												If there are more than 10 (DHP11B) or 64 (DHx41B) parameters to write, declare 
												NUMOF_INITIALPARAMETER in your program.
	
													VAR_GLOBAL CONSTANT
														NUMOF_INITIALPARAMETER : UDINT := 20;	
													END_VAR
	
												##################################################################*)
			-------------------------------------------------------------------------------------------------------------------------------------------------------------
		(* IDs of the PDO telegrams. The IDs are always calculated with the following IDs as a basis + the address of the bus coupler *)

		RxPDO 								ARRAY[1..32] OF MC_PDO_COSLAVE;			(* MOVI-PLC --> Slave *)
												(* := 16#200,16#300,16#400,16#500,16#780,16#240,16#340,16#440,16#540,16#7C0;	*)
		-------------------------------------------------------------------------------------------------------------------------------------------------------------
		TxPDO 								ARRAY[1..32] OF MC_PDO_COSLAVE; 			(* Slave --> MOVI-PLC *)
												(*:= 16#180,16#280,16#380,16#480,16#680,16#1C0,16#2C0,16#3C0,16#4C0,16#6C0;*)
	*)
END_VAR
IF Enable AND NOT Done THEN

	(*########################################################

		Configuration of CANopenSlave (SEW OCC11B)
		
	#########################################################

		TransmissionType for TxPDOs and RxPDOs:

			0:										Event controlled and sychron (with SYNC-Object)
			1-240:									Cyclic and synchron (with SYNC-Object)
			254:									Producer specified
			255:									Acyclic and eventcontrolled 
			255 and EventTime = InhibitTime:	Cyclic

	#########################################################	*)


	(*************************************************** TxPDOs of CANOpenSlave ( MOVI-PLC ReceiveObjects) ***********************************************************)

	ExtConfig.NumberOfTxPDO				:= 4;		(*  TxPDO ---> CANopenSlave Transmit *)

	ExtConfig.TxPDO[1].EventTime			:= 200;		(* Slave: Index 0x18xx SubIndex 5: CycleTime in ms for CANopenSlave TXPDO *)
	ExtConfig.TxPDO[1].InhibitTime			:= 5;		(* Slave: Index 0x18xx SubIndex 3: InhibitTime in ms for CANopenSlave TxPDO *)
	ExtConfig.TxPDO[1].TransmissionType	:= 255;		(* Slave: Index 0x18xx SubIndex 2: TransmissionType for this TxPDO *)

	ExtConfig.TxPDO[2].EventTime			:= 100;		(* Slave: Index 0x18xx SubIndex 5: CycleTime in ms for CANopenSlave TXPDO *)
	ExtConfig.TxPDO[2].InhibitTime			:= 100;		(* Slave: Index 0x18xx SubIndex 3: InhibitTime in ms for CANopenSlave TxPDO *)
	ExtConfig.TxPDO[2].TransmissionType	:= 255;		(* Slave: Index 0x18xx SubIndex 2: TransmissionType for this TxPDO *)

	ExtConfig.TxPDO[3].EventTime			:= 100;		(* Slave: Index 0x18xx SubIndex 5: CycleTime in ms for CANopenSlave TXPDO *)
	ExtConfig.TxPDO[3].InhibitTime			:= 100;		(* Slave: Index 0x18xx SubIndex 3: InhibitTime in ms for CANopenSlave TxPDO *)
	ExtConfig.TxPDO[3].TransmissionType	:= 255;		(* Slave: Index 0x18xx SubIndex 2: TransmissionType for this TxPDO *)

	ExtConfig.TxPDO[4].EventTime			:= 100;		(* Slave: Index 0x18xx SubIndex 5: CycleTime in ms for CANopenSlave TXPDO *)
	ExtConfig.TxPDO[4].InhibitTime			:= 100;		(* Slave: Index 0x18xx SubIndex 3: InhibitTime in ms for CANopenSlave TxPDO *)
	ExtConfig.TxPDO[4].TransmissionType	:= 255;		(* Slave: Index 0x18xx SubIndex 2: TransmissionType for this TxPDO *)


	(*************************************************** RxPDOs of CANOpenSlave ( MOVI-PLC TransmitObjects) **********************************************************)

	ExtConfig.NumberOfRxPDO				:= 4;		(*  RxPDO ---> CANopenSlave Receive *)

	ExtConfig.RxPDO[1].EventTime			:= 200;		(* Master: CycleTime in ms for TransmitObjects (MOVI-PLC) *)
	ExtConfig.RxPDO[1].InhibitTime			:= 5;		(* Master: InhibitTime in ms for TransmitObjects (MOVI-PLC) *)
	ExtConfig.RxPDO[1].Length				:= 1;		(* Master: Length of this TransmitObject in bytes *)
	ExtConfig.RxPDO[1].TransmissionType	:= 255;		(* Slave: Index 0x14xx SubIndex 2: TransmissionType for this RxPDO *)

	ExtConfig.RxPDO[2].EventTime			:= 100;		(* Master: CycleTime in ms for TransmitObjects (MOVI-PLC) *)
	ExtConfig.RxPDO[2].InhibitTime			:= 100;		(* Master: InhibitTime in ms for TransmitObjects (MOVI-PLC) *)
	ExtConfig.RxPDO[2].Length				:= 8;		(* Master: Length of this TransmitObject in bytes *)
	ExtConfig.RxPDO[2].TransmissionType	:= 255;		(* Slave: Index 0x14xx SubIndex 2: TransmissionType for this RxPDO *)

	ExtConfig.RxPDO[3].EventTime			:= 100;		(* Master: CycleTime in ms for TransmitObjects (MOVI-PLC) *)
	ExtConfig.RxPDO[3].InhibitTime			:= 100;		(* Master: InhibitTime in ms for TransmitObjects (MOVI-PLC) *)
	ExtConfig.RxPDO[3].Length				:= 8;		(* Master: Length of this TransmitObject in bytes *)
	ExtConfig.RxPDO[3].TransmissionType	:= 255;		(* Slave: Index 0x14xx SubIndex 2: TransmissionType for this RxPDO *)

	ExtConfig.RxPDO[4].EventTime			:= 100;		(* Master: CycleTime in ms for TransmitObjects (MOVI-PLC) *)
	ExtConfig.RxPDO[4].InhibitTime			:= 100;		(* Master: InhibitTime in ms for TransmitObjects (MOVI-PLC) *)
	ExtConfig.RxPDO[4].Length				:= 8;		(* Master: Length of this TransmitObject in bytes *)
	ExtConfig.RxPDO[4].TransmissionType	:= 255;		(* Slave: Index 0x14xx SubIndex 2: TransmissionType for this RxPDO *)


	(***************************************************** Additional parameters to set in the CANOpenSlave  ***************************************************************)

	(* Enable transmission of analog inputs *)
	ExtConfig.stInitialParameter_COSlave.aIndex[1]			:= 16#6423;
	ExtConfig.stInitialParameter_COSlave.aSubIndex[1]	:= 0;
	ExtConfig.stInitialParameter_COSlave.aBytes[1]		:= 1;
	ExtConfig.stInitialParameter_COSlave.aData[1]			:= 1;


	(********************************************** Additional configuration. Default values are in most cases sufficient *****************************************************)

	ExtConfig.bIOHold						:= FALSE;
	ExtConfig.bNoSettingsDownload			:= FALSE;
	ExtConfig.bWaitBeforeOperational		:= FALSE;
	ExtConfig.bResetUnconditional			:= FALSE;

	ExtConfig.TimeOutHeartBeat				:= 400;				(* [ms] *)
	ExtConfig.TimeOutNodeGuarding		:= 0;				(* [ms]. CAUTION ! DHP11B (MOVI-PLC basic) does NOT support NodeGuarding *)
	ExtConfig.TimeOutInitSequence			:= 10;				(* [seconds]. If the Init-Sequence takes longer than this TimeOut time --> Error *)
	ExtConfig.SyncCOBID						:= 0;				(* SyncObject ID for TransmissionType 0-240 (RxPDO). Usually 16#8000_0080. If 0, the ID will not be written *)
	ExtConfig.SyncTime						:= 0;				(* CycleTime for the SYNC-Object *)

	ExtConfig.SBUSGateway_Address			:= 0(*1001*);			(* OSC71B Address,when used *)

	ExtConfig.TxPDO[1].COBID				:= 16#180;			(* In order to disable the use of RTR frames for the PDOs, set bit 30 = "RTR not allowed" *)
	ExtConfig.TxPDO[2].COBID				:= 16#280;			(* Ex. 16#4000_0280 *)
	ExtConfig.TxPDO[3].COBID				:= 16#380;
	ExtConfig.TxPDO[4].COBID				:= 16#480;			(* NOTE! These values are base values. The input "Address" will automatically be added *)
	ExtConfig.TxPDO[5].COBID				:= 16#680;
	ExtConfig.TxPDO[6].COBID				:= 16#1C0;
	ExtConfig.TxPDO[7].COBID				:= 16#2C0;
	ExtConfig.TxPDO[8].COBID				:= 16#3C0;
	ExtConfig.TxPDO[9].COBID				:= 16#4C0;
	ExtConfig.TxPDO[10].COBID				:= 16#6C0;

	ExtConfig.RxPDO[1].COBID				:= 16#200;
	ExtConfig.RxPDO[2].COBID				:= 16#300;
	ExtConfig.RxPDO[3].COBID				:= 16#400;
	ExtConfig.RxPDO[4].COBID				:= 16#500;
	ExtConfig.RxPDO[5].COBID				:= 16#780;
	ExtConfig.RxPDO[6].COBID				:= 16#240;
	ExtConfig.RxPDO[7].COBID				:= 16#340;
	ExtConfig.RxPDO[8].COBID				:= 16#440;
	ExtConfig.RxPDO[9].COBID				:= 16#540;
	ExtConfig.RxPDO[10].COBID				:= 16#7C0;

	Done := TRUE;

END_IF
END_FUNCTION_BLOCK

(* POU CodeSamples/CANopen/UniversalMaster/FB_Configuration_CANopenSlave_TR_AbsEncoder, ST *)
FUNCTION_BLOCK FB_Configuration_CANopenSlave_TR_AbsEncoder
VAR_INPUT
	Enable: BOOL; 			(* Activate config *)
END_VAR
VAR_OUTPUT
	Done: BOOL;				(* Config done *)
END_VAR
VAR_IN_OUT
	ExtConfig : MC_EXTENDEDCONFIG_COSLAVE	;
	(*
		########################################################################################################
			MC_EXTENDEDCONFIG_COSLAVE
		#########################################################################################################

						
		Variable								Value			Description
		-------------------------------------------------------------------------------------------------------------------------------------------------------------
		bWaitBeforeOperational 				BOOL;			When TRUE, after the coupler has been parameterized, it won't be switched in operational
																before this variable is FALSE. This can be used for example, to store the configuration with the FB
																MPLC_Universal_CANopen, with Service "SEWIOS_STORE", after a reset of the coppler 
		-------------------------------------------------------------------------------------------------------------------------------------------------------------
		bNoSettingsDownload 				BOOL;			TRUE : No configuration of the module. The configuration has to be done manually.
		-------------------------------------------------------------------------------------------------------------------------------------------------------------
		bResetUnconditional 					BOOL;			Even if the Connect FB isn't in fault it is possible to reset the bus coppler
		-------------------------------------------------------------------------------------------------------------------------------------------------------------
		bIOHold 								BOOL;			TRUE : Input data remain unchanged and the output data are not resetet also if the FB is in fault 
		-------------------------------------------------------------------------------------------------------------------------------------------------------------
		TimeOutHeartBeat					UINT;			If this value (ms) is different to zero, HeartbeatMode will be activated
		-------------------------------------------------------------------------------------------------------------------------------------------------------------
		TimeOutNodeGuarding 				UINT;			If this value (ms) is different to zero, NodeGuarding will be activated. 
																Caution ! The MOVI-PLC basic doesn´t support NodeGuarding 
		-------------------------------------------------------------------------------------------------------------------------------------------------------------
		TimeOutInitSequence					UINT;			Timeout for initialisation sequence (seconds) 
		-------------------------------------------------------------------------------------------------------------------------------------------------------------
		NumberOfRxPDO 					UINT;			Receive PDO : MOVI-PLC --> Slave  max. 32 
		-------------------------------------------------------------------------------------------------------------------------------------------------------------
		NumberOfTxPDO 						UINT;			Send PDO :      Slave --> MOVI-PLC  max 32 
		-------------------------------------------------------------------------------------------------------------------------------------------------------------	
		SyncTime 								USINT;			Cycle time of the sync telegram in ms. 
																Default = 0 : no sync will be started.
																If  SyncTime > 0, this FB initializes a sync telegram with the ID set at SyncCOBID. 
																The slave has to support synchronous communication 
		-------------------------------------------------------------------------------------------------------------------------------------------------------------
		SyncCOBID							UINT;			Index 1005h. ID of the sync telegram. Usually 16#80. IF 0, the ID won't be written.
		-------------------------------------------------------------------------------------------------------------------------------------------------------------
		SyncTimeOut 							INT := -1;		Index 1006h. Normally equal to SyncTime. 
																The slave usually set SyncTimeOut equal to SyncTime * 1.5. 
																If < 0, the index won't be written. 0 means no control over the sync interval 
		-------------------------------------------------------------------------------------------------------------------------------------------------------------
		stInitialParameter_COSlave 			MC_INITIALPARAMETER_COSLAVE;
												(*#################################################################
												With this struct, user defined parameters will be written to the BusCoupler after the
												initialization of the MPLC_ConnectUniversalSlave_CANopen. 
												Add the following code to your program to initialise the struct : 
												Example:
												Index 16#6423:	Activates the event-driven transmission of PDOs with analog inputs
												Index 16#3500:	Index from the manufacturer specific profile area
	
													stInitialParameter_COSlave.aIndex[1] := 16#6423;  	(* Index to write to *)
													stInitialParameter_COSlave.aSubIndex[1] := 0;   	(* SubIndex to write to *)
													stInitialParameter_COSlave.aBytes[1] := 1;   		(* Number of bytes to write  *)
													stInitialParameter_COSlave.aData[1] := 1;   			(* Data *)
	
													stInitialParameter_COSlave.aIndex[2] := 16#3500;  	(* Index to write to *)
													stInitialParameter_COSlave.aSubIndex[2] := 0;   	(* SubIndex to write to *)
													stInitialParameter_COSlave.aBytes[2] := 2;   		(* Number of bytes to write *)
													stInitialParameter_COSlave.aData[2] := 5;   			(* Data *)
	
												If there are more than 10 (DHP11B) or 64 (DHx41B) parameters to write, declare 
												NUMOF_INITIALPARAMETER in your program.
	
													VAR_GLOBAL CONSTANT
														NUMOF_INITIALPARAMETER : UDINT := 20;	
													END_VAR
	
												##################################################################*)
			-------------------------------------------------------------------------------------------------------------------------------------------------------------
		(* IDs of the PDO telegrams. The IDs are always calculated with the following IDs as a basis + the address of the bus coupler *)

		RxPDO 								ARRAY[1..32] OF MC_PDO_COSLAVE;			(* MOVI-PLC --> Slave *)
												(* := 16#200,16#300,16#400,16#500,16#780,16#240,16#340,16#440,16#540,16#7C0;	*)
		-------------------------------------------------------------------------------------------------------------------------------------------------------------
		TxPDO 								ARRAY[1..32] OF MC_PDO_COSLAVE; 			(* Slave --> MOVI-PLC *)
												(*:= 16#180,16#280,16#380,16#480,16#680,16#1C0,16#2C0,16#3C0,16#4C0,16#6C0;*)
	*)
END_VAR
IF Enable AND NOT Done THEN

	(*########################################################

		Configuration of CANopenSlave (T+R AbsEncoder)
		
	#########################################################

		TransmissionType for TxPDOs and RxPDOs:

			0:										Event controlled and sychron (with SYNC-Object)
			1-240:									Cyclic and synchron (with SYNC-Object)
			254:									Producer specified
			255:									Acyclic and eventcontrolled 
			255 and EventTime = InhibitTime:	Cyclic

	#########################################################	*)


	(*************************************************** TxPDOs of CANOpenSlave ( MOVI-PLC ReceiveObjects) ***********************************************************)

	ExtConfig.NumberOfTxPDO				:= 1;		(*  TxPDO ---> CANopenSlave Transmit *)

	ExtConfig.TxPDO[1].EventTime			:= 20;		(* Slave: Index 0x18xx SubIndex 5: CycleTime in ms for CANopenSlave TXPDO *)
	ExtConfig.TxPDO[1].InhibitTime			:= 20;		(* Slave: Index 0x18xx SubIndex 3: InhibitTime in ms for CANopenSlave TxPDO *)
	ExtConfig.TxPDO[1].TransmissionType	:= 254;		(* Slave: Index 0x18xx SubIndex 2: TransmissionType for this TxPDO *)


	(*************************************************** RxPDOs of CANOpenSlave ( MOVI-PLC TransmitObjects) **********************************************************)

	ExtConfig.NumberOfRxPDO				:= 0;		(*  RxPDO ---> CANopenSlave Receive *)

	(* ExtConfig.RxPDO[1].EventTime		:= 0;		(* Master: CycleTime in ms for TransmitObjects (MOVI-PLC) *)
	ExtConfig.RxPDO[1].InhibitTime			:= 0;		(* Master: InhibitTime in ms for TransmitObjects (MOVI-PLC) *)
	ExtConfig.RxPDO[1].Length				:= 2;		(* Master: Length of this TransmitObject in bytes *)
	ExtConfig.RxPDO[1].TransmissionType	:= 255;		(* Slave: Index 0x14xx SubIndex 2: TransmissionType for this RxPDO *)*)


	(***************************************************** Additional parameters to set in the CANOpenSlave  ***************************************************************)

	(* Set rotation direction *)
	ExtConfig.stInitialParameter_COSlave.aIndex[1]			:= 16#6000;
	ExtConfig.stInitialParameter_COSlave.aSubIndex[1]	:= 0;
	ExtConfig.stInitialParameter_COSlave.aBytes[1]		:= 2;
	ExtConfig.stInitialParameter_COSlave.aData[1]			:= 0;		(* 0 = CV, 1 = CCV *)

	(* Set cyclic timer for Tx PDO1 *)
	ExtConfig.stInitialParameter_COSlave.aIndex[2]			:= 16#6200;
	ExtConfig.stInitialParameter_COSlave.aSubIndex[2]	:= 0;
	ExtConfig.stInitialParameter_COSlave.aBytes[2]		:= 2;
	ExtConfig.stInitialParameter_COSlave.aData[2]			:= 20;		(* [ms] *)

	(* Write reference offset to AbsEncoder, Index 6003.0, data = new position *)
	(* Write Delivery state to AbsEncoder, Index 1011.1, data = 16#6C_6F_61_64 (load) *)
	(* Save values in Flash memory in the AbsEncoder, Index 1010.1, data = 16#73_61_76_65 (save) *)


	(********************************************** Additional configuration. Default values are in most cases sufficient *****************************************************)

	ExtConfig.bIOHold						:= FALSE;
	ExtConfig.bNoSettingsDownload			:= FALSE;
	ExtConfig.bWaitBeforeOperational		:= FALSE;
	ExtConfig.bResetUnconditional			:= FALSE;

	ExtConfig.TimeOutHeartBeat				:= 0;				(* [ms] *)
	ExtConfig.TimeOutNodeGuarding		:= 400;				(* [ms]. CAUTION ! DHP11B (MOVI-PLC basic) does NOT support NodeGuarding *)
	ExtConfig.TimeOutInitSequence			:= 5;				(* [seconds]. If the Init-Sequence takes longer than this TimeOut time --> Error *)
	ExtConfig.SyncCOBID						:= 0;				(* SyncObject ID for TransmissionType 0-240 (RxPDO). Usually 128. If 0, the ID will not be written *)
	ExtConfig.SyncTime						:= 0;				(* CycleTime for the SYNC-Object *)

	ExtConfig.TxPDO[1].COBID				:= 16#180;			(* In order to disable the use of RTR frames for the PDOs, set bit 30 = "RTR not allowed" *)
	ExtConfig.TxPDO[2].COBID				:= 16#280;			(* Ex. 16#4000_0280 *)
	ExtConfig.TxPDO[3].COBID				:= 16#380;
	ExtConfig.TxPDO[4].COBID				:= 16#480;			(* NOTE! These values are base values. The input "Address" will automatically be added *)
	ExtConfig.TxPDO[5].COBID				:= 16#680;
	ExtConfig.TxPDO[6].COBID				:= 16#1C0;
	ExtConfig.TxPDO[7].COBID				:= 16#2C0;
	ExtConfig.TxPDO[8].COBID				:= 16#3C0;
	ExtConfig.TxPDO[9].COBID				:= 16#4C0;
	ExtConfig.TxPDO[10].COBID				:= 16#6C0;

	ExtConfig.RxPDO[1].COBID				:= 16#200;
	ExtConfig.RxPDO[2].COBID				:= 16#300;
	ExtConfig.RxPDO[3].COBID				:= 16#400;
	ExtConfig.RxPDO[4].COBID				:= 16#500;
	ExtConfig.RxPDO[5].COBID				:= 16#780;
	ExtConfig.RxPDO[6].COBID				:= 16#240;
	ExtConfig.RxPDO[7].COBID				:= 16#340;
	ExtConfig.RxPDO[8].COBID				:= 16#440;
	ExtConfig.RxPDO[9].COBID				:= 16#540;
	ExtConfig.RxPDO[10].COBID				:= 16#7C0;

	Done := TRUE;

END_IF
END_FUNCTION_BLOCK

(* POU CodeSamples/CANopen/UniversalMaster/FB_Configuration_CANopenSlave_Wachendorff, ST *)
FUNCTION_BLOCK FB_Configuration_CANopenSlave_Wachendorff
VAR_INPUT
	Enable: BOOL; 			(* Activate config *)
END_VAR
VAR_OUTPUT
	Done: BOOL;				(* Config done *)
END_VAR
VAR_IN_OUT
	ExtConfig : MC_EXTENDEDCONFIG_COSLAVE	;
	(*
		########################################################################################################
			MC_EXTENDEDCONFIG_COSLAVE
		#########################################################################################################

						
		Variable								Value			Description
		-------------------------------------------------------------------------------------------------------------------------------------------------------------
		bWaitBeforeOperational 				BOOL;			When TRUE, after the coupler has been parameterized, it won't be switched in operational
																before this variable is FALSE. This can be used for example, to store the configuration with the FB
																MPLC_Universal_CANopen, with Service "SEWIOS_STORE", after a reset of the coppler 
		-------------------------------------------------------------------------------------------------------------------------------------------------------------
		bNoSettingsDownload 				BOOL;			TRUE : No configuration of the module. The configuration has to be done manually.
		-------------------------------------------------------------------------------------------------------------------------------------------------------------
		bResetUnconditional 					BOOL;			Even if the Connect FB isn't in fault it is possible to reset the bus coppler
		-------------------------------------------------------------------------------------------------------------------------------------------------------------
		bIOHold 								BOOL;			TRUE : Input data remain unchanged and the output data are not resetet also if the FB is in fault 
		-------------------------------------------------------------------------------------------------------------------------------------------------------------
		TimeOutHeartBeat					UINT;			If this value (ms) is different to zero, HeartbeatMode will be activated

		bNoHeartBeat_Producer:				BOOL := FALSE; (*Index 1017 SubIndex 0 not available *)
		-------------------------------------------------------------------------------------------------------------------------------------------------------------
		TimeOutNodeGuarding 				UINT;			If this value (ms) is different to zero, NodeGuarding will be activated. 
																Caution ! The MOVI-PLC basic doesn´t support NodeGuarding 
	
		bNoNodeGuarding:					BOOL:=FALSE; (* the Index of NodeGuarding isn`t available *)
		-------------------------------------------------------------------------------------------------------------------------------------------------------------
		TimeOutInitSequence					UINT;			Timeout for initialisation sequence (seconds) 
		-------------------------------------------------------------------------------------------------------------------------------------------------------------
		NumberOfRxPDO 					UINT;			Receive PDO : MOVI-PLC --> Slave  max. 32 
		-------------------------------------------------------------------------------------------------------------------------------------------------------------
		NumberOfTxPDO 						UINT;			Send PDO :      Slave --> MOVI-PLC  max 32 
		-------------------------------------------------------------------------------------------------------------------------------------------------------------	
		OffsetOfRxPDO:						UINT;			Offset for the 1. RxPDO
		-------------------------------------------------------------------------------------------------------------------------------------------------------------		
		OffsetOfTxPDO:						UINT;			Offset for the 1. TxPDO
		-------------------------------------------------------------------------------------------------------------------------------------------------------------	
		SyncTime 								USINT;			Cycle time of the sync telegram in ms. 
																Default = 0 : no sync will be started.
																If  SyncTime > 0, this FB initializes a sync telegram with the ID set at SyncCOBID. 
																The slave has to support synchronous communication 
		-------------------------------------------------------------------------------------------------------------------------------------------------------------
		SyncCOBID							UINT;			Index 1005h. ID of the sync telegram. Usually 16#80. IF 0, the ID won't be written.
		-------------------------------------------------------------------------------------------------------------------------------------------------------------
		SyncTimeOut 							INT := -1;		Index 1006h. Normally equal to SyncTime. 
																The slave usually set SyncTimeOut equal to SyncTime * 1.5. 
																If < 0, the index won't be written. 0 means no control over the sync interval 
		-------------------------------------------------------------------------------------------------------------------------------------------------------------
		stInitialParameter_COSlave 			MC_INITIALPARAMETER_COSLAVE;
												(*#################################################################
												With this struct, user defined parameters will be written to the BusCoupler after the
												initialization of the MPLC_ConnectUniversalSlave_CANopen. 
												Add the following code to your program to initialise the struct : 
												Example:
												Index 16#6423:	Activates the event-driven transmission of PDOs with analog inputs
												Index 16#3500:	Index from the manufacturer specific profile area
	
													stInitialParameter_COSlave.aIndex[1] := 16#6423;  	(* Index to write to *)
													stInitialParameter_COSlave.aSubIndex[1] := 0;   	(* SubIndex to write to *)
													stInitialParameter_COSlave.aBytes[1] := 1;   		(* Number of bytes to write  *)
													stInitialParameter_COSlave.aData[1] := 1;   			(* Data *)
	
													stInitialParameter_COSlave.aIndex[2] := 16#3500;  	(* Index to write to *)
													stInitialParameter_COSlave.aSubIndex[2] := 0;   	(* SubIndex to write to *)
													stInitialParameter_COSlave.aBytes[2] := 2;   		(* Number of bytes to write *)
													stInitialParameter_COSlave.aData[2] := 5;   			(* Data *)
	
												If there are more than 10 (DHP11B) or 64 (DHx41B) parameters to write, declare 
												NUMOF_INITIALPARAMETER in your program.
	
													VAR_GLOBAL CONSTANT
														NUMOF_INITIALPARAMETER : UDINT := 20;	
													END_VAR
	
												##################################################################*)

		bNoDeactivatePDO:			BOOL := FALSE; (* Change of Transmission Type, Inhibit- and Event- Time without deactivate RxPDO and TxPDO*)

			-------------------------------------------------------------------------------------------------------------------------------------------------------------
		(* IDs of the PDO telegrams. The IDs are always calculated with the following IDs as a basis + the address of the bus coupler *)

		RxPDO 								ARRAY[1..32] OF MC_PDO_COSLAVE;			(* MOVI-PLC --> Slave *)
												(* := 16#200,16#300,16#400,16#500,16#780,16#240,16#340,16#440,16#540,16#7C0;	*)
		-------------------------------------------------------------------------------------------------------------------------------------------------------------
		TxPDO 								ARRAY[1..32] OF MC_PDO_COSLAVE; 			(* Slave --> MOVI-PLC *)
												(*:= 16#180,16#280,16#380,16#480,16#680,16#1C0,16#2C0,16#3C0,16#4C0,16#6C0;*)
	*)
END_VAR
{library private}
VAR
	fbCANopen_aktiv: CANopen_activ;
	Error: BOOL;
	Error_ID: DINT;
END_VAR
IF Enable AND NOT Done THEN

(*  !!!!!!!  only once TO activate !!!!!!*)
(*
	(*######################################################*)
		(* set Baudrate and CAN-ID *)
	fbCANopen_aktiv(Node:= SBUS_Node_2,
					Address_Default := 60,(* Default Address or old Address 0...127*)
					Address:= 60,(* new Address 1...63*)
					Baudrate:=2, (* 0 = 1 M , 2 = 500 k , 3 = 250 k baud*)
					Error => Error,
					ErrorID=> Error_ID);


		RETURN;
	(*######################################################*)
*)


	(*########################################################

		Configuration of CANopenSlave (Wachendorff AbsEncoder)
		
	#########################################################

		TransmissionType for TxPDOs and RxPDOs:

			0:										Event controlled and sychron (with SYNC-Object)
			1-240:									Cyclic and synchron (with SYNC-Object)
			254:									Producer specified
			255:									Acyclic and eventcontrolled 
			255 and EventTime = InhibitTime:	Cyclic

	#########################################################	*)

(*	ExtConfig.OffsetOfTxPDO := 2;*)
	(*************************************************** TxPDOs of CANOpenSlave ( MOVI-PLC ReceiveObjects) ***********************************************************)

	ExtConfig.NumberOfTxPDO				:= 3;		(*  TxPDO ---> CANopenSlave Transmit *)

	ExtConfig.TxPDO[1].EventTime			:= 20;		(* Slave: Index 0x18xx SubIndex 5: CycleTime in ms for CANopenSlave TXPDO *)
	ExtConfig.TxPDO[1].InhibitTime			:= 10;		(* Slave: Index 0x18xx SubIndex 3: InhibitTime in ms for CANopenSlave TxPDO *)
	ExtConfig.TxPDO[1].TransmissionType	:= 254;		(* Slave: Index 0x18xx SubIndex 2: TransmissionType for this TxPDO *)

	ExtConfig.TxPDO[2].EventTime			:= 0;		(* Slave: Index 0x18xx SubIndex 5: CycleTime in ms for CANopenSlave TXPDO *)
	ExtConfig.TxPDO[2].InhibitTime			:= 0;		(* Slave: Index 0x18xx SubIndex 3: InhibitTime in ms for CANopenSlave TxPDO *)
	ExtConfig.TxPDO[2].TransmissionType	:= 1;		(* Slave: Index 0x18xx SubIndex 2: TransmissionType for this TxPDO *)

	ExtConfig.TxPDO[3].EventTime			:= 0;		(* Slave: Index 0x18xx SubIndex 5: CycleTime in ms for CANopenSlave TXPDO *)
	ExtConfig.TxPDO[3].InhibitTime			:= 0;		(* Slave: Index 0x18xx SubIndex 3: InhibitTime in ms for CANopenSlave TxPDO *)
	ExtConfig.TxPDO[3].TransmissionType	:= 1;		(* Slave: Index 0x18xx SubIndex 2: TransmissionType for this TxPDO *)

	(*************************************************** RxPDOs of CANOpenSlave ( MOVI-PLC TransmitObjects) **********************************************************)

	ExtConfig.NumberOfRxPDO				:= 0;		(*  RxPDO ---> CANopenSlave Receive *)

	(* ExtConfig.RxPDO[1].EventTime		:= 0;		(* Master: CycleTime in ms for TransmitObjects (MOVI-PLC) *)
	ExtConfig.RxPDO[1].InhibitTime			:= 0;		(* Master: InhibitTime in ms for TransmitObjects (MOVI-PLC) *)
	ExtConfig.RxPDO[1].Length				:= 2;		(* Master: Length of this TransmitObject in bytes *)
	ExtConfig.RxPDO[1].TransmissionType	:= 255;		(* Slave: Index 0x14xx SubIndex 2: TransmissionType for this RxPDO *)*)


	(***************************************************** Additional parameters to set in the CANOpenSlave  ***************************************************************)

	(* Set rotation direction *)
	ExtConfig.stInitialParameter_COSlave.aIndex[1]			:= 16#6000;
	ExtConfig.stInitialParameter_COSlave.aSubIndex[1]	:= 0;
	ExtConfig.stInitialParameter_COSlave.aBytes[1]		:= 2;
	ExtConfig.stInitialParameter_COSlave.aData[1]			:= 0;		(* 0 = CV, 1 = CCV *)

(*	(* Set cyclic timer for Tx PDO1 *)
	ExtConfig.stInitialParameter_COSlave.aIndex[2]			:= 16#6200;
	ExtConfig.stInitialParameter_COSlave.aSubIndex[2]	:= 0;
	ExtConfig.stInitialParameter_COSlave.aBytes[2]		:= 2;
	ExtConfig.stInitialParameter_COSlave.aData[2]			:= 20;		(* [ms] *)*)

(* deactivate Tx PDO1 *)
	ExtConfig.stInitialParameter_COSlave.aIndex[2]			:= 16#1800;
	ExtConfig.stInitialParameter_COSlave.aSubIndex[2]	:= 2;
	ExtConfig.stInitialParameter_COSlave.aBytes[2]		:= 1;
	ExtConfig.stInitialParameter_COSlave.aData[2]			:= 16#FF;

	ExtConfig.stInitialParameter_COSlave.aIndex[3]			:= 16#1800;
	ExtConfig.stInitialParameter_COSlave.aSubIndex[3]	:= 5;
	ExtConfig.stInitialParameter_COSlave.aBytes[3]		:= 2;
	ExtConfig.stInitialParameter_COSlave.aData[3]			:= 16#0000;

(* deactivate Tx PDO2 *)
	ExtConfig.stInitialParameter_COSlave.aIndex[4]			:= 16#1801;
	ExtConfig.stInitialParameter_COSlave.aSubIndex[4]	:= 2;
	ExtConfig.stInitialParameter_COSlave.aBytes[4]		:= 1;
	ExtConfig.stInitialParameter_COSlave.aData[4]			:= 16#FF;

	ExtConfig.stInitialParameter_COSlave.aIndex[5]			:= 16#1801;
	ExtConfig.stInitialParameter_COSlave.aSubIndex[5]	:= 5;
	ExtConfig.stInitialParameter_COSlave.aBytes[5]		:= 2;
	ExtConfig.stInitialParameter_COSlave.aData[5]			:= 16#0000;

	(* Write reference offset to AbsEncoder, Index 6003.0, data = new position *)
	(* Write Delivery state to AbsEncoder, Index 1011.1, data = 16#6C_6F_61_64 (load) *)
	(* Save values in Flash memory in the AbsEncoder, Index 1010.1, data = 16#73_61_76_65 (save) *)


	(********************************************** Additional configuration. Default values are in most cases sufficient *****************************************************)

	ExtConfig.bIOHold						:= FALSE;
	ExtConfig.bNoSettingsDownload			:= FALSE;
	ExtConfig.bWaitBeforeOperational		:= FALSE;
	ExtConfig.bResetUnconditional			:= FALSE;

	ExtConfig.TimeOutHeartBeat				:= 400;				(* [ms] *)
	ExtConfig.TimeOutNodeGuarding		:= 0;				(* [ms]. CAUTION ! DHP11B (MOVI-PLC basic) does NOT support NodeGuarding *)
	ExtConfig.TimeOutInitSequence			:= 15;				(* [seconds]. If the Init-Sequence takes longer than this TimeOut time --> Error *)
	ExtConfig.SyncCOBID						:= 128;				(* SyncObject ID for TransmissionType 0-240 (RxPDO). Usually 128. If 0, the ID will not be written *)
	ExtConfig.SyncTime						:= 5;				(* CycleTime for the SYNC-Object *)

	ExtConfig.TxPDO[1].COBID				:= 16#180;			(* In order to disable the use of RTR frames for the PDOs, set bit 30 = "RTR not allowed" *)
	ExtConfig.TxPDO[2].COBID				:= 16#280;			(* Ex. 16#4000_0280 *)
	ExtConfig.TxPDO[3].COBID				:= 16#380;
	ExtConfig.TxPDO[4].COBID				:= 16#480;			(* NOTE! These values are base values. The input "Address" will automatically be added *)
	ExtConfig.TxPDO[5].COBID				:= 16#680;
	ExtConfig.TxPDO[6].COBID				:= 16#1C0;
	ExtConfig.TxPDO[7].COBID				:= 16#2C0;
	ExtConfig.TxPDO[8].COBID				:= 16#3C0;
	ExtConfig.TxPDO[9].COBID				:= 16#4C0;
	ExtConfig.TxPDO[10].COBID				:= 16#6C0;

	ExtConfig.RxPDO[1].COBID				:= 16#200;
	ExtConfig.RxPDO[2].COBID				:= 16#300;
	ExtConfig.RxPDO[3].COBID				:= 16#400;
	ExtConfig.RxPDO[4].COBID				:= 16#500;
	ExtConfig.RxPDO[5].COBID				:= 16#780;
	ExtConfig.RxPDO[6].COBID				:= 16#240;
	ExtConfig.RxPDO[7].COBID				:= 16#340;
	ExtConfig.RxPDO[8].COBID				:= 16#440;
	ExtConfig.RxPDO[9].COBID				:= 16#540;
	ExtConfig.RxPDO[10].COBID				:= 16#7C0;

	Done := TRUE;
END_IF
END_FUNCTION_BLOCK

(* POU CodeSamples/CANopen/UniversalMaster/FB_Configuration_CANopenSlave_WAGO_750_337, ST *)
FUNCTION_BLOCK FB_Configuration_CANopenSlave_WAGO_750_337
VAR_INPUT
	Enable: BOOL; 			(* Activate config *)
END_VAR
VAR_OUTPUT
	Done: BOOL;				(* Config done *)
END_VAR
VAR_IN_OUT
	ExtConfig : MC_EXTENDEDCONFIG_COSLAVE	;
	(*
		########################################################################################################
			MC_EXTENDEDCONFIG_COSLAVE
		#########################################################################################################

						
		Variable								Value			Description
		-------------------------------------------------------------------------------------------------------------------------------------------------------------
		bWaitBeforeOperational 				BOOL;			When TRUE, after the coupler has been parameterized, it won't be switched in operational
																before this variable is FALSE. This can be used for example, to store the configuration with the FB
																MPLC_Universal_CANopen, with Service "SEWIOS_STORE", after a reset of the coppler 
		-------------------------------------------------------------------------------------------------------------------------------------------------------------
		bNoSettingsDownload 				BOOL;			TRUE : No configuration of the module. The configuration has to be done manually.
		-------------------------------------------------------------------------------------------------------------------------------------------------------------
		bResetUnconditional 					BOOL;			Even if the Connect FB isn't in fault it is possible to reset the bus coppler
		-------------------------------------------------------------------------------------------------------------------------------------------------------------
		bIOHold 								BOOL;			TRUE : Input data remain unchanged and the output data are not resetet also if the FB is in fault 
		-------------------------------------------------------------------------------------------------------------------------------------------------------------
		TimeOutHeartBeat					UINT;			If this value (ms) is different to zero, HeartbeatMode will be activated
		-------------------------------------------------------------------------------------------------------------------------------------------------------------
		TimeOutNodeGuarding 				UINT;			If this value (ms) is different to zero, NodeGuarding will be activated. 
																Caution ! The MOVI-PLC basic doesn´t support NodeGuarding 
		-------------------------------------------------------------------------------------------------------------------------------------------------------------
		TimeOutInitSequence					UINT;			Timeout for initialisation sequence (seconds) 
		-------------------------------------------------------------------------------------------------------------------------------------------------------------
		NumberOfRxPDO 					UINT;			Receive PDO : MOVI-PLC --> Slave  max. 32 
		-------------------------------------------------------------------------------------------------------------------------------------------------------------
		NumberOfTxPDO 						UINT;			Send PDO :      Slave --> MOVI-PLC  max 32 
		-------------------------------------------------------------------------------------------------------------------------------------------------------------	
		SyncTime 								USINT;			Cycle time of the sync telegram in ms. 
																Default = 0 : no sync will be started.
																If  SyncTime > 0, this FB initializes a sync telegram with the ID set at SyncCOBID. 
																The slave has to support synchronous communication 
		-------------------------------------------------------------------------------------------------------------------------------------------------------------
		SyncCOBID							UINT;			Index 1005h. ID of the sync telegram. Usually 16#80. IF 0, the ID won't be written.
		-------------------------------------------------------------------------------------------------------------------------------------------------------------
		SyncTimeOut 							INT := -1;		Index 1006h. Normally equal to SyncTime. 
																The slave usually set SyncTimeOut equal to SyncTime * 1.5. 
																If < 0, the index won't be written. 0 means no control over the sync interval 
		-------------------------------------------------------------------------------------------------------------------------------------------------------------
		stInitialParameter_COSlave 			MC_INITIALPARAMETER_COSLAVE;
												(*#################################################################
												With this struct, user defined parameters will be written to the BusCoupler after the
												initialization of the MPLC_ConnectUniversalSlave_CANopen. 
												Add the following code to your program to initialise the struct : 
												Example:
												Index 16#6423:	Activates the event-driven transmission of PDOs with analog inputs
												Index 16#3500:	Index from the manufacturer specific profile area
	
													stInitialParameter_COSlave.aIndex[1] := 16#6423;  	(* Index to write to *)
													stInitialParameter_COSlave.aSubIndex[1] := 0;   	(* SubIndex to write to *)
													stInitialParameter_COSlave.aBytes[1] := 1;   		(* Number of bytes to write  *)
													stInitialParameter_COSlave.aData[1] := 1;   			(* Data *)
	
													stInitialParameter_COSlave.aIndex[2] := 16#3500;  	(* Index to write to *)
													stInitialParameter_COSlave.aSubIndex[2] := 0;   	(* SubIndex to write to *)
													stInitialParameter_COSlave.aBytes[2] := 2;   		(* Number of bytes to write *)
													stInitialParameter_COSlave.aData[2] := 5;   			(* Data *)
	
												If there are more than 10 (DHP11B) or 64 (DHx41B) parameters to write, declare 
												NUMOF_INITIALPARAMETER in your program.
	
													VAR_GLOBAL CONSTANT
														NUMOF_INITIALPARAMETER : UDINT := 20;	
													END_VAR
	
												##################################################################*)
			-------------------------------------------------------------------------------------------------------------------------------------------------------------
		(* IDs of the PDO telegrams. The IDs are always calculated with the following IDs as a basis + the address of the bus coupler *)

		RxPDO 								ARRAY[1..32] OF MC_PDO_COSLAVE;			(* MOVI-PLC --> Slave *)
												(* := 16#200,16#300,16#400,16#500,16#780,16#240,16#340,16#440,16#540,16#7C0;	*)
		-------------------------------------------------------------------------------------------------------------------------------------------------------------
		TxPDO 								ARRAY[1..32] OF MC_PDO_COSLAVE; 			(* Slave --> MOVI-PLC *)
												(*:= 16#180,16#280,16#380,16#480,16#680,16#1C0,16#2C0,16#3C0,16#4C0,16#6C0;*)
	*)
END_VAR
IF Enable AND NOT Done THEN

	(*########################################################

		Configuration of CANopenSlave (WAGO 750-337)
		
	#########################################################

		TransmissionType for TxPDOs and RxPDOs:

			0:										Event controlled and sychron (with SYNC-Object)
			1-240:									Cyclic and synchron (with SYNC-Object)
			254:									Producer specified
			255:									Acyclic and eventcontrolled 
			255 and EventTime = InhibitTime:	Cyclic

	#########################################################	*)


	(*************************************************** TxPDOs of CANOpenSlave ( MOVI-PLC ReceiveObjects) ***********************************************************)

	ExtConfig.NumberOfTxPDO				:= 2;		(*  TxPDO ---> CANopenSlave Transmit *)

	ExtConfig.TxPDO[1].EventTime			:= 200;		(* Slave: Index 0x18xx SubIndex 5: CycleTime in ms for CANopenSlave TXPDO *)
	ExtConfig.TxPDO[1].InhibitTime			:= 5;		(* Slave: Index 0x18xx SubIndex 3: InhibitTime in ms for CANopenSlave TxPDO *)
	ExtConfig.TxPDO[1].TransmissionType	:= 255;		(* Slave: Index 0x18xx SubIndex 2: TransmissionType for this TxPDO *)

	ExtConfig.TxPDO[2].EventTime			:= 100;		(* Slave: Index 0x18xx SubIndex 5: CycleTime in ms for CANopenSlave TXPDO *)
	ExtConfig.TxPDO[2].InhibitTime			:= 100;		(* Slave: Index 0x18xx SubIndex 3: InhibitTime in ms for CANopenSlave TxPDO *)
	ExtConfig.TxPDO[2].TransmissionType	:= 255;		(* Slave: Index 0x18xx SubIndex 2: TransmissionType for this TxPDO *)


	(*************************************************** RxPDOs of CANOpenSlave ( MOVI-PLC TransmitObjects) **********************************************************)

	ExtConfig.NumberOfRxPDO				:= 2;		(*  RxPDO ---> CANopenSlave Receive *)

	ExtConfig.RxPDO[1].EventTime			:= 200;		(* Master: CycleTime in ms for TransmitObjects (MOVI-PLC) *)
	ExtConfig.RxPDO[1].InhibitTime			:= 5;		(* Master: InhibitTime in ms for TransmitObjects (MOVI-PLC) *)
	ExtConfig.RxPDO[1].Length				:= 8;		(* Master: Length of this TransmitObject in bytes *)
	ExtConfig.RxPDO[1].TransmissionType	:= 255;		(* Slave: Index 0x14xx SubIndex 2: TransmissionType for this RxPDO *)

	ExtConfig.RxPDO[2].EventTime			:= 100;		(* Master: CycleTime in ms for TransmitObjects (MOVI-PLC) *)
	ExtConfig.RxPDO[2].InhibitTime			:= 100;		(* Master: InhibitTime in ms for TransmitObjects (MOVI-PLC) *)
	ExtConfig.RxPDO[2].Length				:= 8;		(* Master: Length of this TransmitObject in bytes *)
	ExtConfig.RxPDO[2].TransmissionType	:= 255;		(* Slave: Index 0x14xx SubIndex 2: TransmissionType for this RxPDO *)


	(***************************************************** Additional parameters to set in the CANOpenSlave  ***************************************************************)

	(* Enable transmission of analog inputs *)
	ExtConfig.stInitialParameter_COSlave.aIndex[1]			:= 16#6423;
	ExtConfig.stInitialParameter_COSlave.aSubIndex[1]	:= 0;
	ExtConfig.stInitialParameter_COSlave.aBytes[1]		:= 1;
	ExtConfig.stInitialParameter_COSlave.aData[1]			:= 1;


	(********************************************** Additional configuration. Default values are in most cases sufficient *****************************************************)

	ExtConfig.bIOHold						:= FALSE;
	ExtConfig.bNoSettingsDownload			:= FALSE;
	ExtConfig.bWaitBeforeOperational		:= FALSE;
	ExtConfig.bResetUnconditional			:= FALSE;

	ExtConfig.TimeOutHeartBeat				:= 400;				(* [ms] *)
	ExtConfig.TimeOutNodeGuarding		:= 0;				(* [ms]. CAUTION ! DHP11B (MOVI-PLC basic) does NOT support NodeGuarding *)
	ExtConfig.TimeOutInitSequence			:= 10;				(* [seconds]. If the Init-Sequence takes longer than this TimeOut time --> Error *)
	ExtConfig.SyncCOBID						:= 0;				(* SyncObject ID for TransmissionType 0-240 (RxPDO). Usually 128. If 0, the ID will not be written *)
	ExtConfig.SyncTime						:= 0;				(* CycleTime for the SYNC-Object *)

	ExtConfig.TxPDO[1].COBID				:= 16#180;			(* In order to disable the use of RTR frames for the PDOs, set bit 30 = "RTR not allowed" *)
	ExtConfig.TxPDO[2].COBID				:= 16#280;			(* Ex. 16#4000_0280 *)
	ExtConfig.TxPDO[3].COBID				:= 16#380;
	ExtConfig.TxPDO[4].COBID				:= 16#480;			(* NOTE! These values are base values. The input "Address" will automatically be added *)
	ExtConfig.TxPDO[5].COBID				:= 16#680;
	ExtConfig.TxPDO[6].COBID				:= 16#1C0;
	ExtConfig.TxPDO[7].COBID				:= 16#2C0;
	ExtConfig.TxPDO[8].COBID				:= 16#3C0;
	ExtConfig.TxPDO[9].COBID				:= 16#4C0;
	ExtConfig.TxPDO[10].COBID				:= 16#6C0;

	ExtConfig.RxPDO[1].COBID				:= 16#200;
	ExtConfig.RxPDO[2].COBID				:= 16#300;
	ExtConfig.RxPDO[3].COBID				:= 16#400;
	ExtConfig.RxPDO[4].COBID				:= 16#500;
	ExtConfig.RxPDO[5].COBID				:= 16#780;
	ExtConfig.RxPDO[6].COBID				:= 16#240;
	ExtConfig.RxPDO[7].COBID				:= 16#340;
	ExtConfig.RxPDO[8].COBID				:= 16#440;
	ExtConfig.RxPDO[9].COBID				:= 16#540;
	ExtConfig.RxPDO[10].COBID				:= 16#7C0;

	Done := TRUE;

END_IF
END_FUNCTION_BLOCK
